SUBAPPLICATION Uebung_006e1 (* SR-Flip-Flop mit 2x IX *)
  (* Standard: 61499-2; Description: Copyright (c) 2023 Meisterschulen am Ostbahnhof This program and the accompanying materials are made available under the terms of the Eclipse Public License 2.0 which is available at https://www.eclipse.org/legal/epl-2.0/ SPDX-License-Identifier: EPL-2.0 *)
  (* Version 1.0, 2023-10-23, Franz Höpfinger, Meisterschulen am Ostbahnhof, initial API and implementation and/or initial documentation *)
  PACKAGE Uebungen;
  IMPORT logiBUS::io::DI::logiBUS_DI::Input_I1;
  IMPORT logiBUS::io::DI::logiBUS_DI::Input_I2;
  IMPORT logiBUS::io::DQ::logiBUS_DO::Output_Q1;
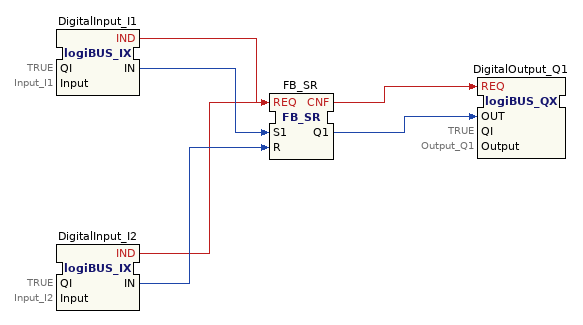
  FBS
    DigitalOutput_Q1 : logiBUS::io::DQ::logiBUS_QX(QI := TRUE, Output := Output_Q1);
    DigitalInput_I1 : logiBUS::io::DI::logiBUS_IX(QI := TRUE, Input := Input_I1);
    DigitalInput_I2 : logiBUS::io::DI::logiBUS_IX(QI := TRUE, Input := Input_I2);
    FB_SR : iec61131::bistableElements::FB_SR;
  END_FBS
  EVENT_CONNECTIONS
    FB_SR.CNF TO DigitalOutput_Q1.REQ;
    DigitalInput_I2.IND TO FB_SR.REQ;
    DigitalInput_I1.IND TO FB_SR.REQ;
  END_CONNECTIONS
  DATA_CONNECTIONS
    FB_SR.Q1 TO DigitalOutput_Q1.OUT;
    DigitalInput_I1.IN TO FB_SR.S1;
    DigitalInput_I2.IN TO FB_SR.R;
  END_CONNECTIONS
END_SUBAPPLICATION
